Yaskawa INFORM job: R1-HOME.JBI

/JOB
//NAME R1-HOME
///FOLDERNAME FOLDER001
//POS
///NPOS 1,1,0,0,0,0
///TOOL 0
///POSTYPE ROBOT
///RECTAN
///RCONF 0,0,0,0,0,0,0,0,0,0,0,0,0,0,0,0,0,0,0,0,0,0,0,0
C00000=1043.998,19.972,-681.753,-3.2675,-33.1665,3.5966
BC00000=539.760,0.026,840.907
//INST
///DATE 2023/07/10 15:23
///ATTR SC,RW,RJ
////FRAME ROBOT
///GROUP1 RB1,BS1
NOP
MOVJ C00000 BC00000 VJ=30.00
END
